(* Schneider Machine Expert - Basic project cel2_teste, file version 3.0.0.0 *)
(* ProjectInformations: Name=Novo projeto *)

HARDWARE
  Cpu 0: TM221CE16T
  ModuleExtensionObject 0: TM3DI16/G
  ModuleExtensionObject 1: TM3DQ16T/G
  ModuleExtensionObject 2: TM3DM8R/G
  ModuleExtensionObject 3: TM3DM8R/G
  ModuleExtensionObject 4: TM3DM8R/G
  ModuleExtensionObject 5: TM3SAF5R/G
  ModuleExtensionObject 6: TM3SAF5R/G
  EthernetConfiguration: NetworkName=M221, IpAllocationMode=FixedAddress, IpAddress=192.168.0.49, SubnetMask=255.255.255.0
  SerialLineConfiguration: Baud=Baud19200, Parity=ParityEven, DataBits=DataBits8, StopBits=StopBits1, PhysicalMedium=PhysicalMediumRs485, TransmissionMode=TransmissionModeModbusRtu, SlaveId=1, Addressing=SlaveAddressing
  MastTask: UsePeriodScanMode=false, PeriodScan=100
  FastTask: Period=255, FastTaskSubroutine=robo - clp
  CpuBehavior: StartingMode=StartAsPreviousState, AutoSaveRamOnEeprom=true, WatchdogPeriod=250

SYMBOLS  (address, symbol, comment, settings)
  %QWN300.9.0:X0 BIT1_SCADA
  %QWN300.9.0:X1 BIT2_SCADA
  %QWN300.9.0:X2 BIT3_SCADA
  %M0       M0  "primeiro paso - ligar celula"
  %M1       M1
  %M2       M2
  %M3       M3
  %M4       M4
  %M5       M5
  %M6       M6
  %M7       M7
  %M8       M8
  %M9       M9
  %M10      M10
  %M11      M11
  %M12      M12
  %M13      M13
  %M14      M14
  %M15      M15
  %M16      M16
  %M17      M17
  %M18      M18
  %M19      M19
  %M20      M20
  %M21      M21
  %M24      DESLIGA_BRANCO
  %M25      DESLIGA_CINZA
  %M26      DESLIGA_CINZA_ESCURO
  %M27      DESLIGA_PRETO
  %M28      DESLIGA_TRANSPARENTE
  %M32      ROBO_BRANCO
  %M33      ROBO_CINZA
  %M34      ROBO_CINZA_ESCURO
  %M35      ROBO_PRETO
  %M36      ROBO_TRANSPARENTE
  %M37      SCADA_SENSORESTEIRA
  %KW0      BASE_BRANCO  [Value=5]
  %KW1      BASE_CINZA  [Value=6]
  %KW2      BASE_CINZA_ESCURO  [Value=7]
  %KW3      BASE_PRETA  [Value=8]
  %KW4      BASE_TRANSPARENTE  [Value=9]
  %TM0      TIMER1  [Preset=4, Base=OneSecond]
  %TM1      TIMER2  [Preset=2, Base=OneSecond, IsRetentive=true]
  %TM2      TIMER3  [Preset=2, Base=OneSecond]
  %TM3      TIMER4  [Preset=2, Base=OneSecond]
  %TM4      TIMER5  [Preset=2, Base=OneSecond]
  %TM5      TIMER6  [Preset=2, Base=OneSecond]
  %TM6      TIMER7  [Preset=2, Base=OneSecond]
  %TM7      TIMER8  [Preset=5, Base=TenMilliSeconds]
  %TM8      TIMER9  [Preset=2, Base=OneSecond]
  %TM9      TIMER10  [Preset=2, Base=OneSecond]
  %TM10     TIMER11  [Preset=2, Base=OneSecond]
  %TM11     TIMER12  [Preset=2, Base=OneSecond]
  %TM12     TIMER13  [Preset=2, Base=OneSecond]
  %TM13     TIMERDESLIGA  [Preset=4, Base=OneSecond]
  %TM14     TIMERDESLIGA2  [Preset=4, Base=OneSecond]
  %TM15     TIMERDESLIGA3  [Preset=4, Base=OneSecond]
  %TM16     TIMERÚLTIMO  [Preset=4, Base=OneSecond]
  %TM17     TIMER17  [Preset=4, Base=OneSecond]
  %TM18     TIMER18  [Preset=2, Base=OneSecond]
  %TM19     TIMER19  [Preset=2, Base=OneSecond]
  %TM20     TIMER20  [Preset=2, Base=OneSecond]
  %TM21     TIMER21  [Preset=3, Base=OneSecond]
  %TM22     TIMER22  [Preset=2, Base=OneSecond]
  %TM23     TIMER23  [Preset=2, Base=OneSecond]
  %TM24       [Preset=1, Base=OneSecond]
  %TM25       [Preset=1, Base=OneSecond]
  %I0.0     RESET
  %I0.1     START_
  %I0.2     STOP
  %I0.3     PECA_ESTEIRA  "Sesnsor que detecta peçpa na garra na esteira"
  %I0.4     AVANCO_TRANSPARENTE  "Sensor Avanço Atuador Base Cinza Escuro"
  %I0.5     AVANCO_BRANCO  "Sensor Avanço Atuador Base Cinza"
  %I0.6     AVANCO_CINZA  "Sensor Avanço Atuador Base Transparente"
  %I0.7     AVANCO_CINZA_ESCURO  "Sensor Avanço Atuador Base Branco"
  %I0.8     AVANCO_PRETA  "Sensor Avanço Atuador Base Preta"
  %Q0.0     DISPENSER_PRETA  "Válvula Dispenser Preta"
  %Q0.1     DISPENSER_CINZA_ESCURO  "Válvula Dispenser Cinza escuro"
  %Q0.2     DISPENSER_CINZA  "Válvula Dispenser cinza claro"
  %Q0.3     DISPENSER_BRANCO  "Válvula Dispenser Branco"
  %Q0.4     DISPENSER_TRANSPARENTE  "Válvula Dispenser Transparente"
  %Q0.5     ATUADOR_X  "Válvula Atuador Eixo X"
  %Q0.6     ATUADOR_Z  "Válvula Atuador Eixo Z"
  %IN301.0.0   "Start forçado para a grob"  [Channel=START]
  %IN301.1.0   "Branco forçado GROB"  [Channel=BRANCO]
  %QN300.2.0 VENTOSA_SCADA  [Channel=NX3008_ventosa]
  %QN300.4.0   [Channel=NX3008_garra]
  %QN300.6.0 ATUADORX_SCADA  [Channel=NX3008_atuador_x]
  %QN300.7.0 ATUADORZ_SCADA  [Channel=NX3008_atuador_z]
  %IWN300.0.0 BASE_MODBUS  [Channel=NX3008_id_base]
  %IWN301.2.0 BASES_GROB  [Channel=Teste_bases]
  %QWN300.1.0   [Channel=NX3008_sensores]
  %QWN300.3.0   [Channel=NX3008_dispensers]
  %QWN300.5.0   [Channel=NX3008_sensor_garra_esteira]
  %QWN300.8.0 CORES  [Channel=NX3008_cores]
  %QWN300.9.0   [Channel=NX3008_Infos_robo]
  %I1.0     RECUOX  "sensor de recuo x"
  %I1.1     AVANCOX  "sensor de avanco x"
  %I1.2     RECUOZ  "sensor de recuo z"
  %I1.3     AVANCOZ  "sesnor de avanco z"
  %I1.4     GARRAABERTA  "sensor da garra aberta do atuador"
  %I1.5     SAIDADISPENSER  "sensor de presenca de saida do dispenser na garra do robo"
  %I1.6     GARRAABROB  "sensor de garra aberta do robo"
  %I1.14    OUTPUT1_VACUO
  %I1.15    OUTPUT2_RBG
  %Q2.0     ATUADORGARRA  "valvula da garra do atuador"
  %Q2.1     GARRAROB
  %Q2.3     VENTOSA_
  %I3.0     ENTRADA1  "modolo de io do robo sem enderecamento"
  %I3.1     ENTRADA2  "modolo de io do robo sem enderecamento"
  %I3.2     ROBOFINALIZADO
  %I3.3     LUZAMARELA
  %Q3.0     BIT1  "modolo de io do robo sem enderecamento"
  %Q3.1     BIT2  "modolo de io do robo sem enderecamento"
  %Q3.2     BIT3  "modolo de io do robo sem enderecamento"
  %I4.0       "Sensor de Recuo Eixo X - celula"
  %I4.1       "Sensor de Avanço Eixo X - esteira"
  %I4.2       "Sensor de Recuo Eixo Z - cima"
  %I4.3       "Sensor de Avanço Eixo Z - baixo"
  %Q4.0       "robo"
  %Q4.1       "robo"
  %Q4.2       "robo"
  %Q4.3       "robo"
  %I5.0       "Sensor de Garra Aberta"
  %I5.1       "Sensor de Peça Montagem"
  %I5.2       "Sensor de Presença Saida do Dispenser"
  %Q5.1       "Válvula Atuador Garra"
  %Q5.2       "vacuum generator"
  %Q5.3       "TORRE DE SINALIZAÇÃO"
  %I6.0     SA_OUTPUTON  "Saída de segurança ligada"
  %I6.1     SA_SUPPLY  "Fornecimento disponível (A1/A2)"
  %I6.2     SA_SUPPLYFAIL  "Fornecimento fora de tolerância"
  %I6.3     SA_CH1  "Canal 1 ativo"
  %I6.4     SA_CH2  "Canal 2 ativo"
  %I6.5     SA_START  "Início ativo"
  %I6.6     SA_K1  "Relé K1 ativado"
  %I6.7     SA_K2  "Relé k2 ativado"
  %I6.8       "Reserved"
  %I6.9     SA_S1  "S1 ativo"
  %I6.10    SA_S2  "S2 ativo"
  %I6.11    SA_S4  "S4 ativo"
  %I6.12    SA_WAITINGFORSTART  "Aguardando por condição de início"
  %I6.13      "Reserved"
  %Q6.0     SA_ENABLE  "Ativação das saídas de segurança habilitada"
  %Q6.1     SA_RESETMODULE  "Módulo de desativação (fonte atual desligada)"
  %Q6.2     SA_KEEPALIVE  "Função de segurança permanece ativa mesmo quando o barramento está 'inativo' (tempo esgotado)"
  %Q6.3       "Reserved"
  %I7.0     SA_OUTPUTON_0  "Saída de segurança ligada"
  %I7.1     SA_SUPPLY_0  "Fornecimento disponível (A1/A2)"
  %I7.2     SA_SUPPLYFAIL_0  "Fornecimento fora de tolerância"
  %I7.3     SA_CH1_0  "Canal 1 ativo"
  %I7.4     SA_CH2_0  "Canal 2 ativo"
  %I7.5     SA_START_0  "Início ativo"
  %I7.6     SA_K1_0  "Relé K1 ativado"
  %I7.7     SA_K2_0  "Relé k2 ativado"
  %I7.8       "Reserved"
  %I7.9     SA_S1_0  "S1 ativo"
  %I7.10    SA_S2_0  "S2 ativo"
  %I7.11    SA_S4_0  "S4 ativo"
  %I7.12    SA_WAITINGFORSTART_0  "Aguardando por condição de início"
  %I7.13      "Reserved"
  %Q7.0     SA_ENABLE_0  "Ativação das saídas de segurança habilitada"
  %Q7.1     SA_RESETMODULE_0  "Módulo de desativação (fonte atual desligada)"
  %Q7.2     SA_KEEPALIVE_0  "Função de segurança permanece ativa mesmo quando o barramento está 'inativo' (tempo esgotado)"
  %Q7.3       "Reserved"

POU Transferencia-SCADA
  (* SectionNumber=1 *)

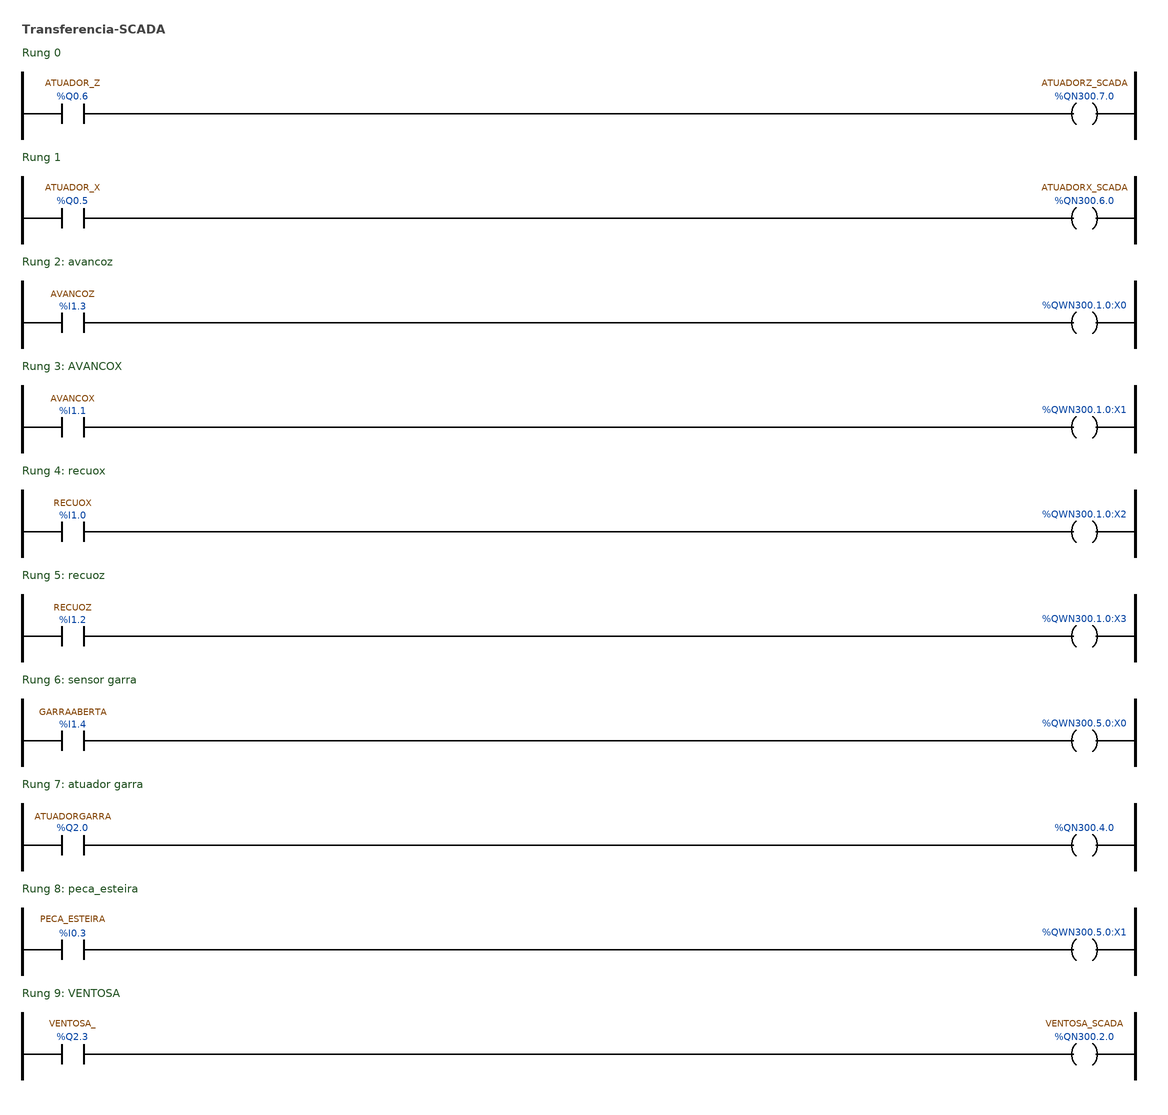

// Rung 0
  LD %Q0.6                (* ATUADOR_Z *)
  ST %QN300.7.0           (* ATUADORZ_SCADA *)
  // as ST:
  //   ATUADORZ_SCADA := ATUADOR_Z;

// Rung 1
  LD %Q0.5                (* ATUADOR_X *)
  ST %QN300.6.0           (* ATUADORX_SCADA *)
  // as ST:
  //   ATUADORX_SCADA := ATUADOR_X;

// Rung 2: avancoz
  LD %I1.3                (* AVANCOZ *)
  ST %QWN300.1.0:X0
  // as ST:
  //   %QWN300.1.0:X0 := AVANCOZ;

// Rung 3: AVANCOX
  LD %I1.1                (* AVANCOX *)
  ST %QWN300.1.0:X1
  // as ST:
  //   %QWN300.1.0:X1 := AVANCOX;

// Rung 4: recuox
  LD %I1.0                (* RECUOX *)
  ST %QWN300.1.0:X2
  // as ST:
  //   %QWN300.1.0:X2 := RECUOX;

// Rung 5: recuoz
  LD %I1.2                (* RECUOZ *)
  ST %QWN300.1.0:X3
  // as ST:
  //   %QWN300.1.0:X3 := RECUOZ;

// Rung 6: sensor garra
  LD %I1.4                (* GARRAABERTA *)
  ST %QWN300.5.0:X0
  // as ST:
  //   %QWN300.5.0:X0 := GARRAABERTA;

// Rung 7: atuador garra
  LD %Q2.0                (* ATUADORGARRA *)
  ST %QN300.4.0
  // as ST:
  //   %QN300.4.0 := ATUADORGARRA;

// Rung 8: peca_esteira
  LD %I0.3                (* PECA_ESTEIRA *)
  ST %QWN300.5.0:X1
  // as ST:
  //   %QWN300.5.0:X1 := PECA_ESTEIRA;

// Rung 9: VENTOSA
  LD %Q2.3                (* VENTOSA_ *)
  ST %QN300.2.0           (* VENTOSA_SCADA *)
  // as ST:
  //   VENTOSA_SCADA := VENTOSA_;

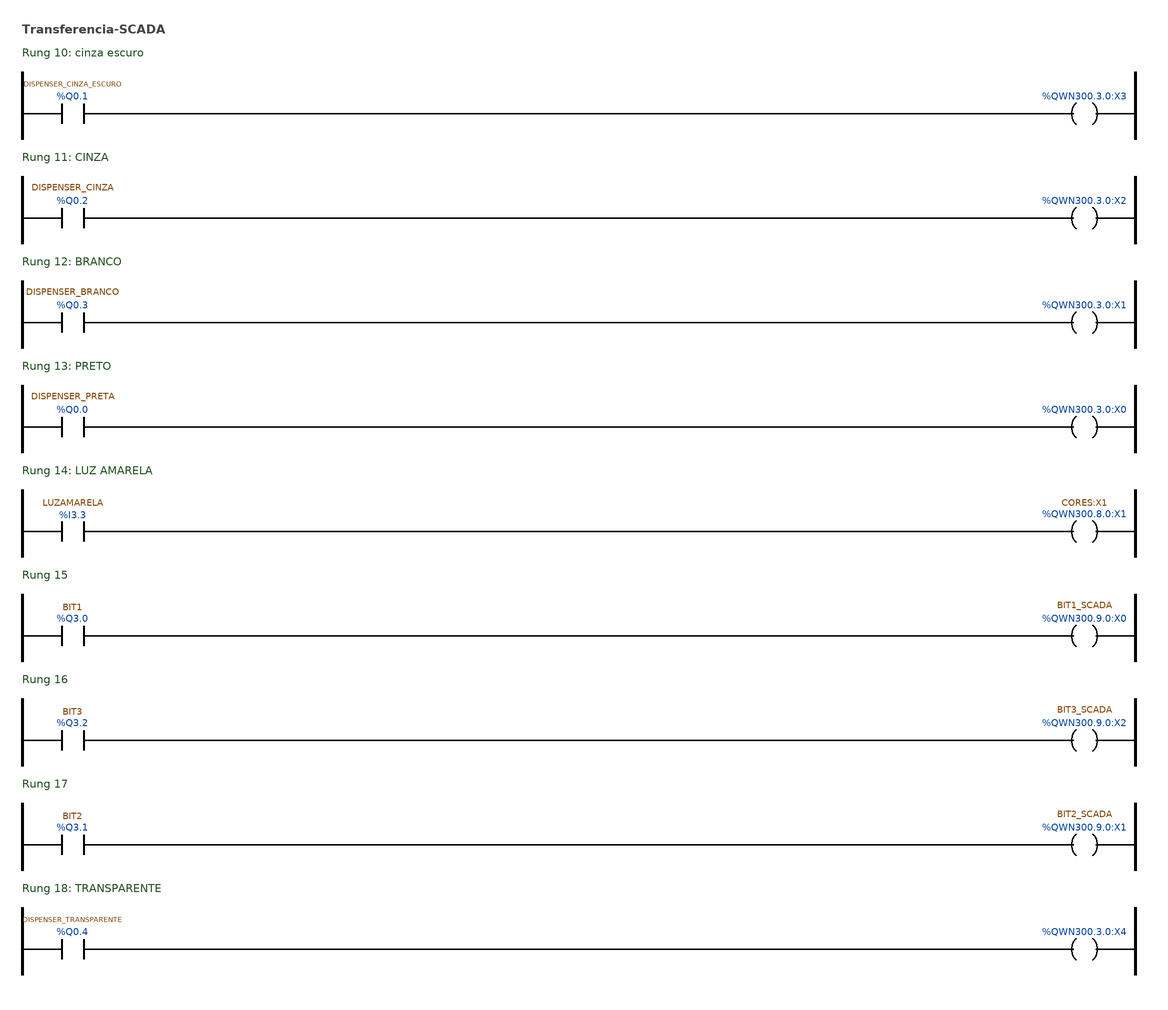

// Rung 10: cinza escuro
  LD %Q0.1                (* DISPENSER_CINZA_ESCURO *)
  ST %QWN300.3.0:X3
  // as ST:
  //   %QWN300.3.0:X3 := DISPENSER_CINZA_ESCURO;

// Rung 11: CINZA
  LD %Q0.2                (* DISPENSER_CINZA *)
  ST %QWN300.3.0:X2
  // as ST:
  //   %QWN300.3.0:X2 := DISPENSER_CINZA;

// Rung 12: BRANCO
  LD %Q0.3                (* DISPENSER_BRANCO *)
  ST %QWN300.3.0:X1
  // as ST:
  //   %QWN300.3.0:X1 := DISPENSER_BRANCO;

// Rung 13: PRETO
  LD %Q0.0                (* DISPENSER_PRETA *)
  ST %QWN300.3.0:X0
  // as ST:
  //   %QWN300.3.0:X0 := DISPENSER_PRETA;

// Rung 14: LUZ AMARELA
  LD %I3.3                (* LUZAMARELA *)
  ST %QWN300.8.0:X1       (* CORES *)
  // as ST:
  //   CORES:X1 := LUZAMARELA;

// Rung 15
  LD %Q3.0                (* BIT1 *)
  ST %QWN300.9.0:X0
  // as ST:
  //   %QWN300.9.0:X0 := BIT1;

// Rung 16
  LD %Q3.2                (* BIT3 *)
  ST %QWN300.9.0:X2
  // as ST:
  //   %QWN300.9.0:X2 := BIT3;

// Rung 17
  LD %Q3.1                (* BIT2 *)
  ST %QWN300.9.0:X1
  // as ST:
  //   %QWN300.9.0:X1 := BIT2;

// Rung 18: TRANSPARENTE
  LD %Q0.4                (* DISPENSER_TRANSPARENTE *)
  ST %QWN300.3.0:X4
  // as ST:
  //   %QWN300.3.0:X4 := DISPENSER_TRANSPARENTE;

POU celula 2
  (* SectionNumber=2 *)

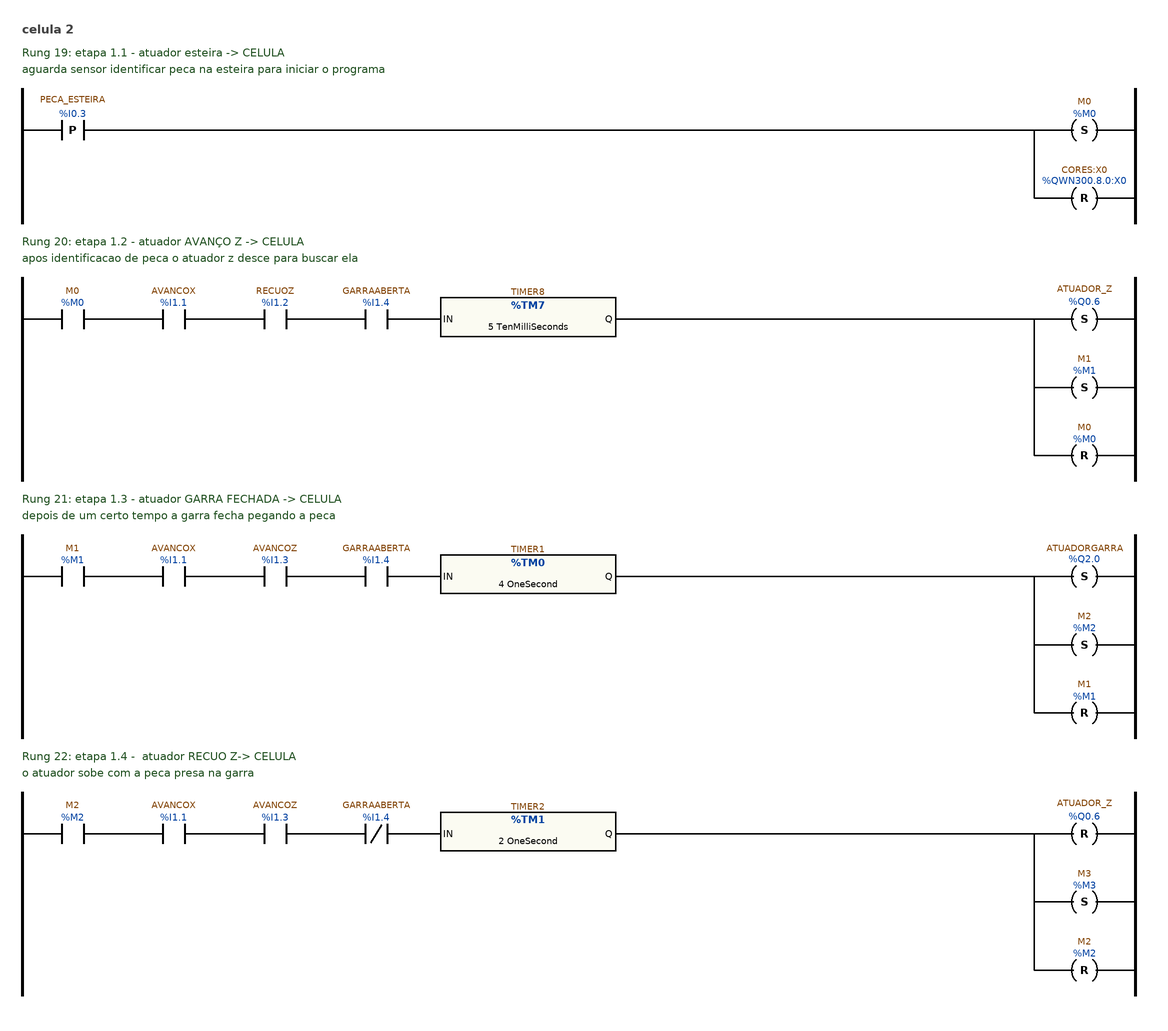

// Rung 19: etapa 1.1 - atuador esteira -> CELULA
// aguarda sensor identificar peca na esteira para iniciar o programa
  LDR %I0.3               (* PECA_ESTEIRA *)
  S %M0                   (* M0 *)
  R %QWN300.8.0:X0        (* CORES *)
  // as ST:
  //   IF RISING(PECA_ESTEIRA) THEN M0 := TRUE; END_IF;
  //   IF RISING(PECA_ESTEIRA) THEN CORES:X0 := FALSE; END_IF;

// Rung 20: etapa 1.2 - atuador AVANÇO Z -> CELULA
// apos identificacao de peca o atuador z desce para buscar ela
  BLK %TM7                (* TIMER8 *)
  LD %M0                  (* M0 *)
  AND %I1.1               (* AVANCOX *)
  AND %I1.2               (* RECUOZ *)
  AND %I1.4               (* GARRAABERTA *)
  IN
  OUT_BLK
  LD Q
  S %Q0.6                 (* ATUADOR_Z *)
  S %M1                   (* M1 *)
  R %M0                   (* M0 *)
  END_BLK
  // as ST:
  //   TIMER8(IN := M0 AND AVANCOX AND RECUOZ AND GARRAABERTA);
  //   IF TIMER8.Q THEN ATUADOR_Z := TRUE; END_IF;
  //   IF TIMER8.Q THEN M1 := TRUE; END_IF;
  //   IF TIMER8.Q THEN M0 := FALSE; END_IF;

// Rung 21: etapa 1.3 - atuador GARRA FECHADA -> CELULA
// depois de um certo tempo a garra fecha pegando a peca
  BLK %TM0                (* TIMER1 *)
  LD %M1                  (* M1 *)
  AND %I1.1               (* AVANCOX *)
  AND %I1.3               (* AVANCOZ *)
  AND %I1.4               (* GARRAABERTA *)
  IN
  OUT_BLK
  LD Q
  S %Q2.0                 (* ATUADORGARRA *)
  S %M2                   (* M2 *)
  R %M1                   (* M1 *)
  END_BLK
  // as ST:
  //   TIMER1(IN := M1 AND AVANCOX AND AVANCOZ AND GARRAABERTA);
  //   IF TIMER1.Q THEN ATUADORGARRA := TRUE; END_IF;
  //   IF TIMER1.Q THEN M2 := TRUE; END_IF;
  //   IF TIMER1.Q THEN M1 := FALSE; END_IF;

// Rung 22: etapa 1.4 -  atuador RECUO Z-> CELULA
// o atuador sobe com a peca presa na garra
  BLK %TM1                (* TIMER2 *)
  LD %M2                  (* M2 *)
  AND %I1.1               (* AVANCOX *)
  AND %I1.3               (* AVANCOZ *)
  ANDN %I1.4              (* GARRAABERTA *)
  IN
  OUT_BLK
  LD Q
  R %Q0.6                 (* ATUADOR_Z *)
  S %M3                   (* M3 *)
  R %M2                   (* M2 *)
  END_BLK
  // as ST:
  //   TIMER2(IN := M2 AND AVANCOX AND AVANCOZ AND NOT GARRAABERTA);
  //   IF TIMER2.Q THEN ATUADOR_Z := FALSE; END_IF;
  //   IF TIMER2.Q THEN M3 := TRUE; END_IF;
  //   IF TIMER2.Q THEN M2 := FALSE; END_IF;

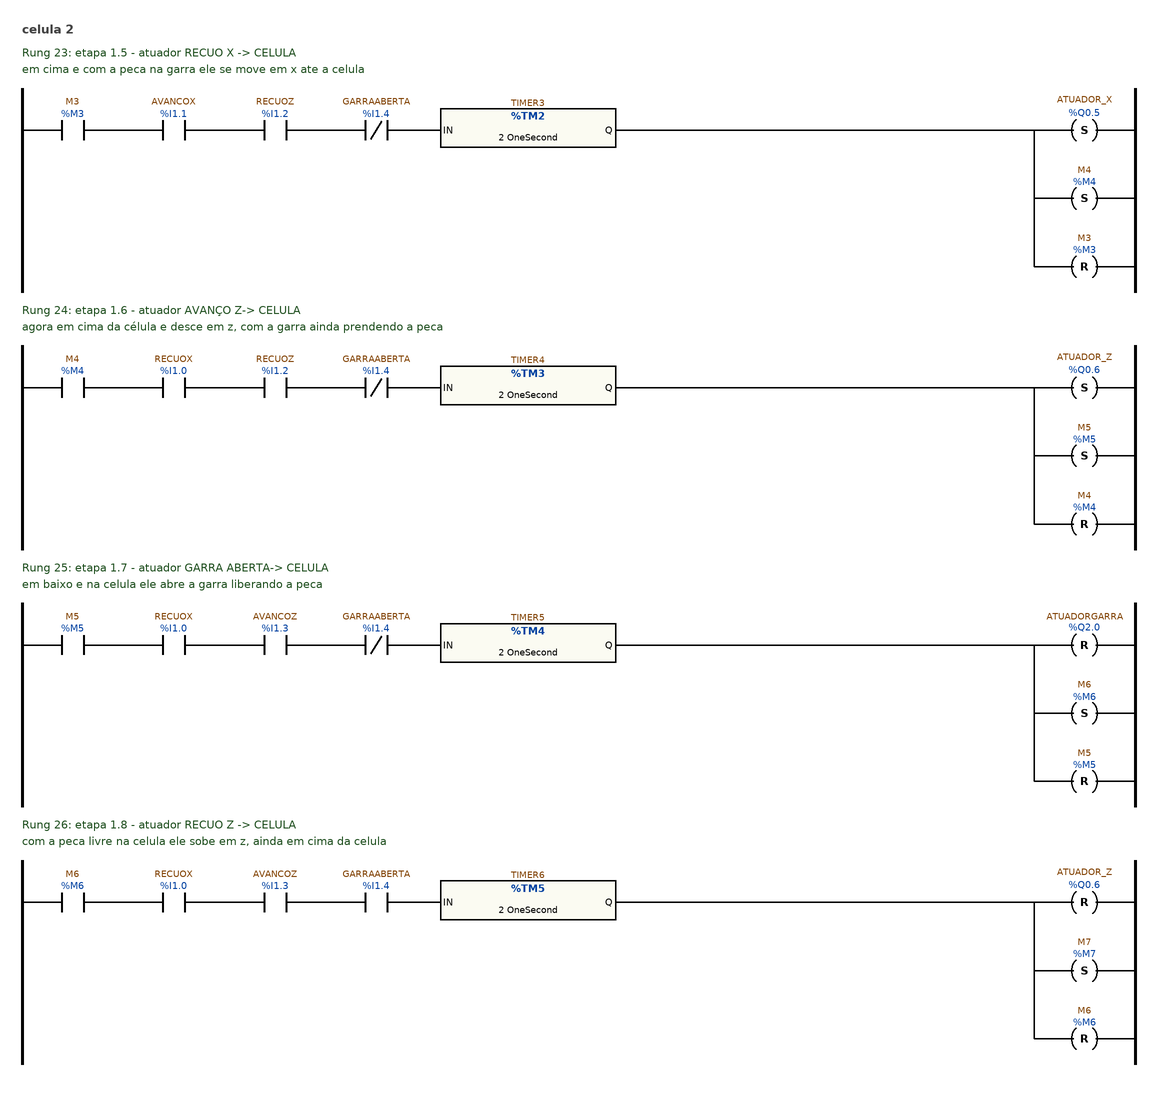

// Rung 23: etapa 1.5 - atuador RECUO X -> CELULA
// em cima e com a peca na garra ele se move em x ate a celula
  BLK %TM2                (* TIMER3 *)
  LD %M3                  (* M3 *)
  AND %I1.1               (* AVANCOX *)
  AND %I1.2               (* RECUOZ *)
  ANDN %I1.4              (* GARRAABERTA *)
  IN
  OUT_BLK
  LD Q
  S %Q0.5                 (* ATUADOR_X *)
  S %M4                   (* M4 *)
  R %M3                   (* M3 *)
  END_BLK
  // as ST:
  //   TIMER3(IN := M3 AND AVANCOX AND RECUOZ AND NOT GARRAABERTA);
  //   IF TIMER3.Q THEN ATUADOR_X := TRUE; END_IF;
  //   IF TIMER3.Q THEN M4 := TRUE; END_IF;
  //   IF TIMER3.Q THEN M3 := FALSE; END_IF;

// Rung 24: etapa 1.6 - atuador AVANÇO Z-> CELULA
// agora em cima da célula e desce em z, com a garra ainda prendendo a peca
  BLK %TM3                (* TIMER4 *)
  LD %M4                  (* M4 *)
  AND %I1.0               (* RECUOX *)
  AND %I1.2               (* RECUOZ *)
  ANDN %I1.4              (* GARRAABERTA *)
  IN
  OUT_BLK
  LD Q
  S %Q0.6                 (* ATUADOR_Z *)
  S %M5                   (* M5 *)
  R %M4                   (* M4 *)
  END_BLK
  // as ST:
  //   TIMER4(IN := M4 AND RECUOX AND RECUOZ AND NOT GARRAABERTA);
  //   IF TIMER4.Q THEN ATUADOR_Z := TRUE; END_IF;
  //   IF TIMER4.Q THEN M5 := TRUE; END_IF;
  //   IF TIMER4.Q THEN M4 := FALSE; END_IF;

// Rung 25: etapa 1.7 - atuador GARRA ABERTA-> CELULA
// em baixo e na celula ele abre a garra liberando a peca
  BLK %TM4                (* TIMER5 *)
  LD %M5                  (* M5 *)
  AND %I1.0               (* RECUOX *)
  AND %I1.3               (* AVANCOZ *)
  ANDN %I1.4              (* GARRAABERTA *)
  IN
  OUT_BLK
  LD Q
  R %Q2.0                 (* ATUADORGARRA *)
  S %M6                   (* M6 *)
  R %M5                   (* M5 *)
  END_BLK
  // as ST:
  //   TIMER5(IN := M5 AND RECUOX AND AVANCOZ AND NOT GARRAABERTA);
  //   IF TIMER5.Q THEN ATUADORGARRA := FALSE; END_IF;
  //   IF TIMER5.Q THEN M6 := TRUE; END_IF;
  //   IF TIMER5.Q THEN M5 := FALSE; END_IF;

// Rung 26: etapa 1.8 - atuador RECUO Z -> CELULA
// com a peca livre na celula ele sobe em z, ainda em cima da celula
  BLK %TM5                (* TIMER6 *)
  LD %M6                  (* M6 *)
  AND %I1.0               (* RECUOX *)
  AND %I1.3               (* AVANCOZ *)
  AND %I1.4               (* GARRAABERTA *)
  IN
  OUT_BLK
  LD Q
  R %Q0.6                 (* ATUADOR_Z *)
  S %M7                   (* M7 *)
  R %M6                   (* M6 *)
  END_BLK
  // as ST:
  //   TIMER6(IN := M6 AND RECUOX AND AVANCOZ AND GARRAABERTA);
  //   IF TIMER6.Q THEN ATUADOR_Z := FALSE; END_IF;
  //   IF TIMER6.Q THEN M7 := TRUE; END_IF;
  //   IF TIMER6.Q THEN M6 := FALSE; END_IF;

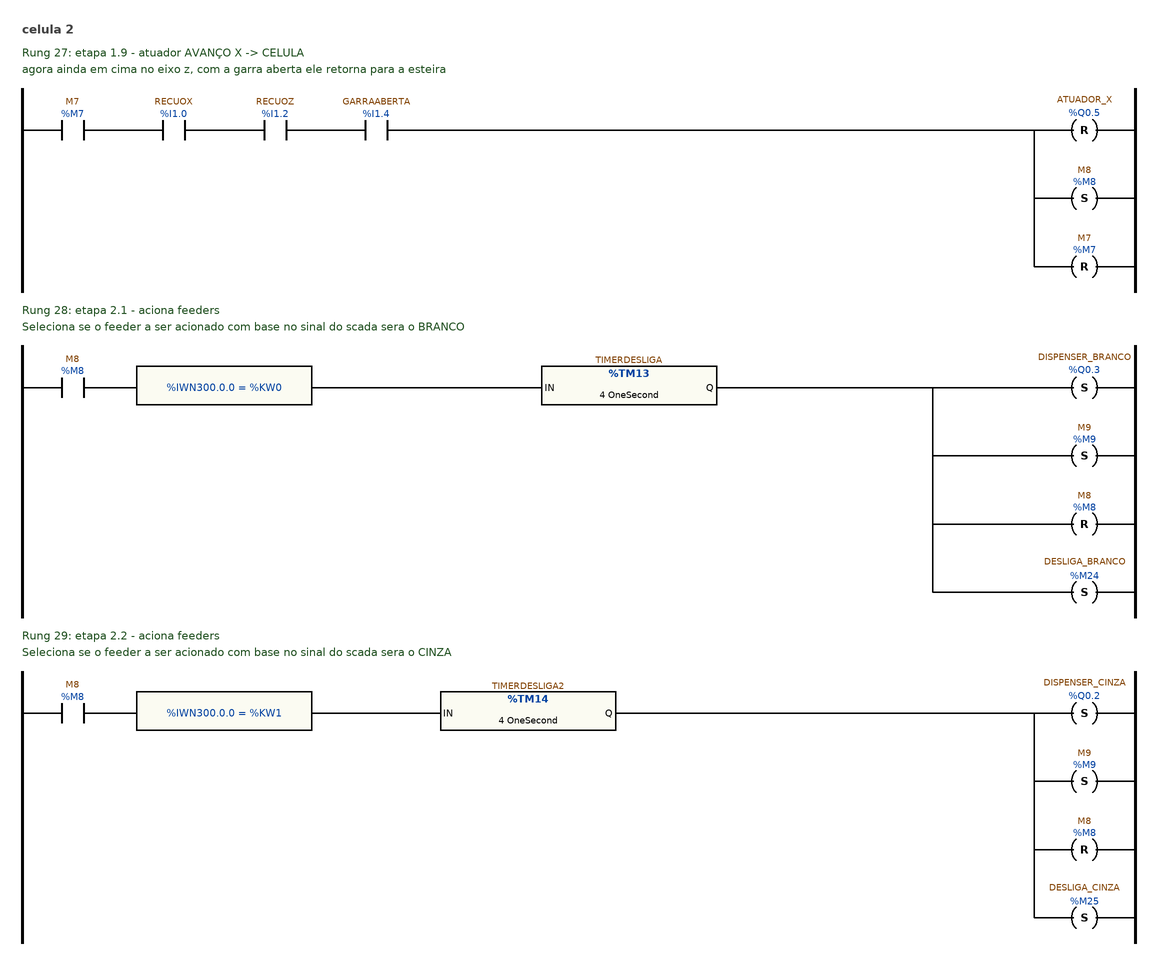

// Rung 27: etapa 1.9 - atuador AVANÇO X -> CELULA
// agora ainda em cima no eixo z, com a garra aberta ele retorna para a esteira
  LD %M7                  (* M7 *)
  AND %I1.0               (* RECUOX *)
  AND %I1.2               (* RECUOZ *)
  AND %I1.4               (* GARRAABERTA *)
  R %Q0.5                 (* ATUADOR_X *)
  S %M8                   (* M8 *)
  R %M7                   (* M7 *)
  // as ST:
  //   IF M7 AND RECUOX AND RECUOZ AND GARRAABERTA THEN ATUADOR_X := FALSE; END_IF;
  //   IF M7 AND RECUOX AND RECUOZ AND GARRAABERTA THEN M8 := TRUE; END_IF;
  //   IF M7 AND RECUOX AND RECUOZ AND GARRAABERTA THEN M7 := FALSE; END_IF;

// Rung 28: etapa 2.1 - aciona feeders
// Seleciona se o feeder a ser acionado com base no sinal do scada sera o BRANCO
  BLK %TM13               (* TIMERDESLIGA *)
  LD %M8                  (* M8 *)
  AND [ %IWN300.0.0 = %KW0 ](* BASE_MODBUS, BASE_BRANCO *)
  IN
  OUT_BLK
  LD Q
  S %Q0.3                 (* DISPENSER_BRANCO *)
  S %M9                   (* M9 *)
  R %M8                   (* M8 *)
  S %M24                  (* DESLIGA_BRANCO *)
  END_BLK
  // as ST:
  //   TIMERDESLIGA(IN := M8 AND BASE_MODBUS = BASE_BRANCO);
  //   IF TIMERDESLIGA.Q THEN DISPENSER_BRANCO := TRUE; END_IF;
  //   IF TIMERDESLIGA.Q THEN M9 := TRUE; END_IF;
  //   IF TIMERDESLIGA.Q THEN M8 := FALSE; END_IF;
  //   IF TIMERDESLIGA.Q THEN DESLIGA_BRANCO := TRUE; END_IF;

// Rung 29: etapa 2.2 - aciona feeders
// Seleciona se o feeder a ser acionado com base no sinal do scada sera o CINZA
  BLK %TM14               (* TIMERDESLIGA2 *)
  LD %M8                  (* M8 *)
  AND [ %IWN300.0.0 = %KW1 ](* BASE_MODBUS, BASE_CINZA *)
  IN
  OUT_BLK
  LD Q
  S %Q0.2                 (* DISPENSER_CINZA *)
  S %M9                   (* M9 *)
  R %M8                   (* M8 *)
  S %M25                  (* DESLIGA_CINZA *)
  END_BLK
  // as ST:
  //   TIMERDESLIGA2(IN := M8 AND BASE_MODBUS = BASE_CINZA);
  //   IF TIMERDESLIGA2.Q THEN DISPENSER_CINZA := TRUE; END_IF;
  //   IF TIMERDESLIGA2.Q THEN M9 := TRUE; END_IF;
  //   IF TIMERDESLIGA2.Q THEN M8 := FALSE; END_IF;
  //   IF TIMERDESLIGA2.Q THEN DESLIGA_CINZA := TRUE; END_IF;

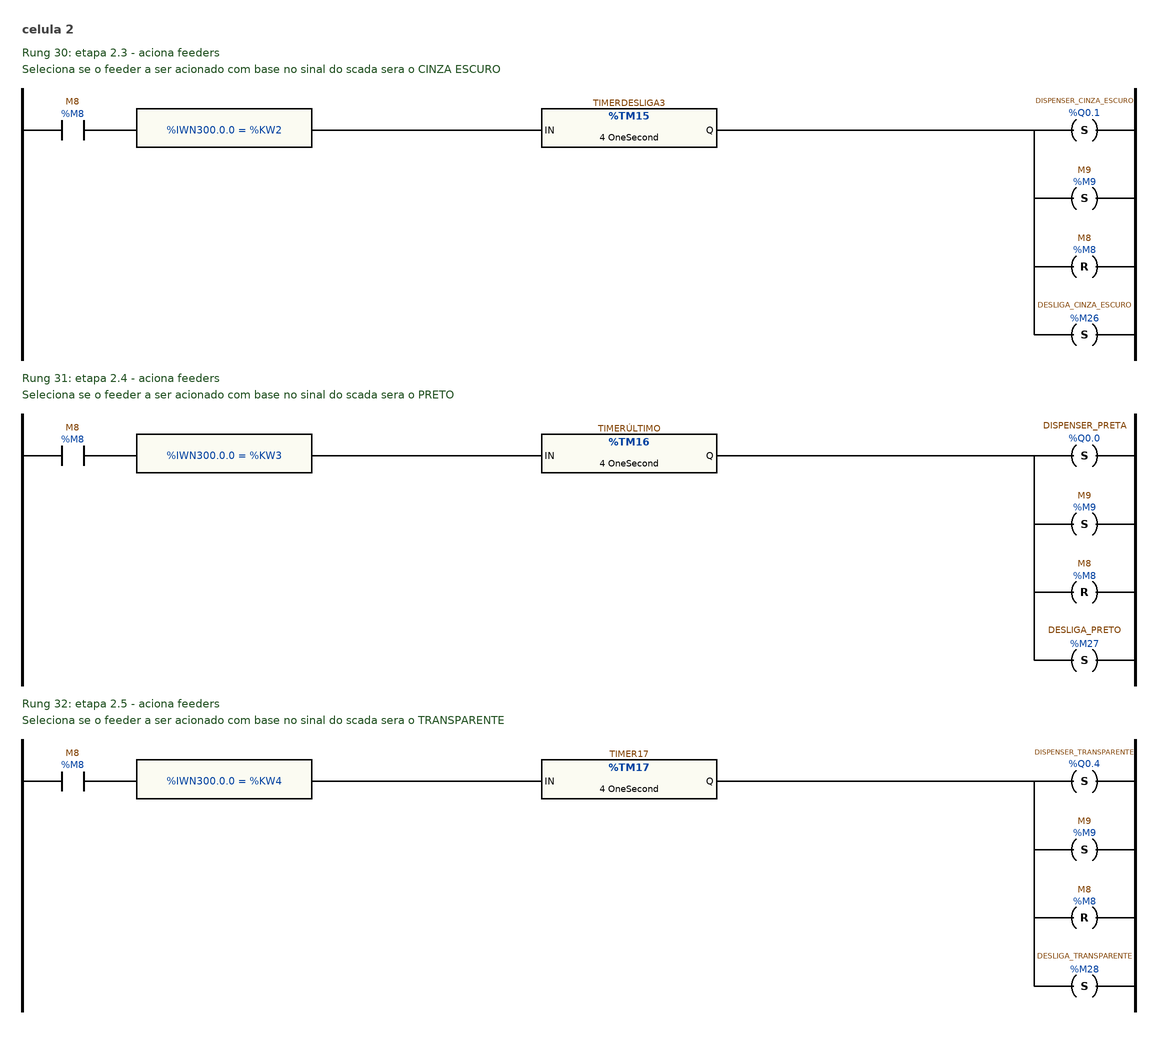

// Rung 30: etapa 2.3 - aciona feeders
// Seleciona se o feeder a ser acionado com base no sinal do scada sera o CINZA ESCURO
  BLK %TM15               (* TIMERDESLIGA3 *)
  LD %M8                  (* M8 *)
  AND [ %IWN300.0.0 = %KW2 ](* BASE_MODBUS, BASE_CINZA_ESCURO *)
  IN
  OUT_BLK
  LD Q
  S %Q0.1                 (* DISPENSER_CINZA_ESCURO *)
  S %M9                   (* M9 *)
  R %M8                   (* M8 *)
  S %M26                  (* DESLIGA_CINZA_ESCURO *)
  END_BLK
  // as ST:
  //   TIMERDESLIGA3(IN := M8 AND BASE_MODBUS = BASE_CINZA_ESCURO);
  //   IF TIMERDESLIGA3.Q THEN DISPENSER_CINZA_ESCURO := TRUE; END_IF;
  //   IF TIMERDESLIGA3.Q THEN M9 := TRUE; END_IF;
  //   IF TIMERDESLIGA3.Q THEN M8 := FALSE; END_IF;
  //   IF TIMERDESLIGA3.Q THEN DESLIGA_CINZA_ESCURO := TRUE; END_IF;

// Rung 31: etapa 2.4 - aciona feeders
// Seleciona se o feeder a ser acionado com base no sinal do scada sera o PRETO
  BLK %TM16               (* TIMERÚLTIMO *)
  LD %M8                  (* M8 *)
  AND [ %IWN300.0.0 = %KW3 ](* BASE_MODBUS, BASE_PRETA *)
  IN
  OUT_BLK
  LD Q
  S %Q0.0                 (* DISPENSER_PRETA *)
  S %M9                   (* M9 *)
  R %M8                   (* M8 *)
  S %M27                  (* DESLIGA_PRETO *)
  END_BLK
  // as ST:
  //   TIMERÚLTIMO(IN := M8 AND BASE_MODBUS = BASE_PRETA);
  //   IF TIMERÚLTIMO.Q THEN DISPENSER_PRETA := TRUE; END_IF;
  //   IF TIMERÚLTIMO.Q THEN M9 := TRUE; END_IF;
  //   IF TIMERÚLTIMO.Q THEN M8 := FALSE; END_IF;
  //   IF TIMERÚLTIMO.Q THEN DESLIGA_PRETO := TRUE; END_IF;

// Rung 32: etapa 2.5 - aciona feeders
// Seleciona se o feeder a ser acionado com base no sinal do scada sera o TRANSPARENTE
  BLK %TM17               (* TIMER17 *)
  LD %M8                  (* M8 *)
  AND [ %IWN300.0.0 = %KW4 ](* BASE_MODBUS, BASE_TRANSPARENTE *)
  IN
  OUT_BLK
  LD Q
  S %Q0.4                 (* DISPENSER_TRANSPARENTE *)
  S %M9                   (* M9 *)
  R %M8                   (* M8 *)
  S %M28                  (* DESLIGA_TRANSPARENTE *)
  END_BLK
  // as ST:
  //   TIMER17(IN := M8 AND BASE_MODBUS = BASE_TRANSPARENTE);
  //   IF TIMER17.Q THEN DISPENSER_TRANSPARENTE := TRUE; END_IF;
  //   IF TIMER17.Q THEN M9 := TRUE; END_IF;
  //   IF TIMER17.Q THEN M8 := FALSE; END_IF;
  //   IF TIMER17.Q THEN DESLIGA_TRANSPARENTE := TRUE; END_IF;

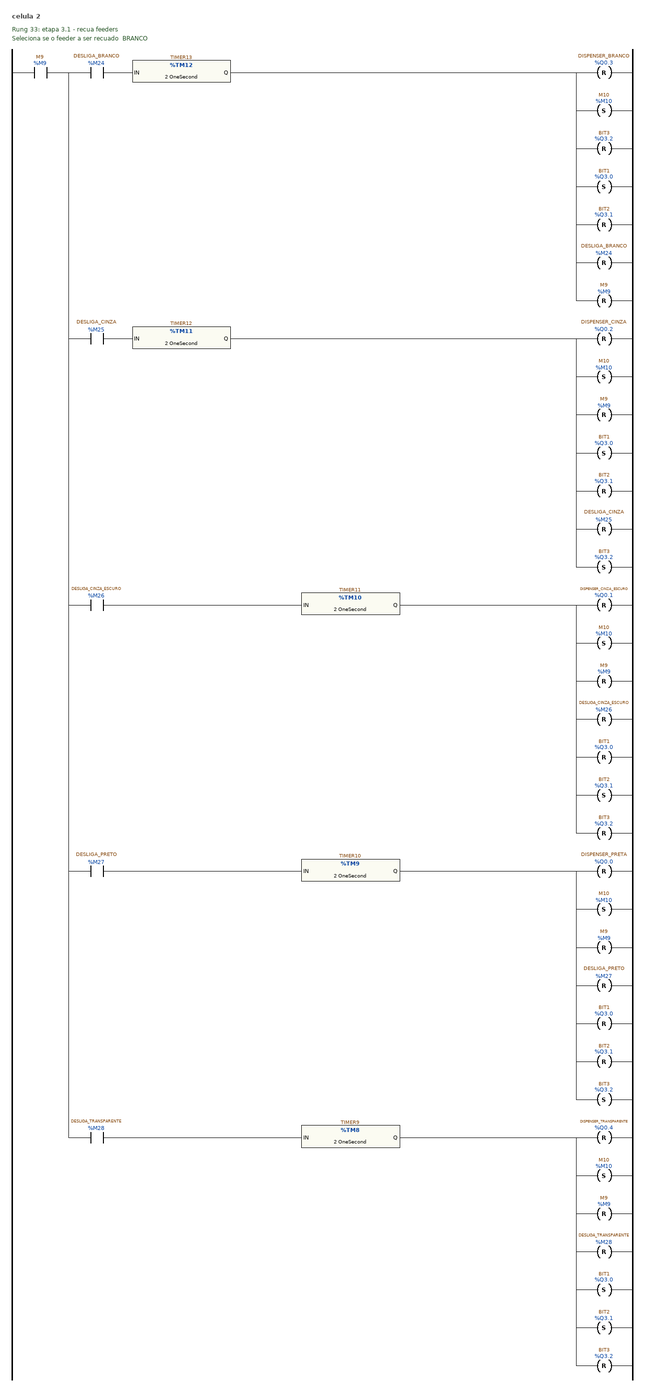

// Rung 33: etapa 3.1 - recua feeders
// Seleciona se o feeder a ser recuado  BRANCO
  LD 1
  MULTIFB
  LD 1
  AND %M9                 (* M9 *)
  ST %MW2009:X0
  BLK %TM12               (* TIMER13 *)
  LD %MW2009:X0
  AND %M24                (* DESLIGA_BRANCO *)
  IN
  OUT_BLK
  LD Q
  R %Q0.3                 (* DISPENSER_BRANCO *)
  S %M10                  (* M10 *)
  R %Q3.2                 (* BIT3 *)
  S %Q3.0                 (* BIT1 *)
  R %Q3.1                 (* BIT2 *)
  R %M24                  (* DESLIGA_BRANCO *)
  R %M9                   (* M9 *)
  END_BLK
  BLK %TM11               (* TIMER12 *)
  LD %MW2009:X0
  AND %M25                (* DESLIGA_CINZA *)
  IN
  OUT_BLK
  LD Q
  R %Q0.2                 (* DISPENSER_CINZA *)
  S %M10                  (* M10 *)
  R %M9                   (* M9 *)
  S %Q3.0                 (* BIT1 *)
  R %Q3.1                 (* BIT2 *)
  R %M25                  (* DESLIGA_CINZA *)
  S %Q3.2                 (* BIT3 *)
  END_BLK
  BLK %TM10               (* TIMER11 *)
  LD %MW2009:X0
  AND %M26                (* DESLIGA_CINZA_ESCURO *)
  IN
  OUT_BLK
  LD Q
  R %Q0.1                 (* DISPENSER_CINZA_ESCURO *)
  S %M10                  (* M10 *)
  R %M9                   (* M9 *)
  R %M26                  (* DESLIGA_CINZA_ESCURO *)
  R %Q3.0                 (* BIT1 *)
  S %Q3.1                 (* BIT2 *)
  R %Q3.2                 (* BIT3 *)
  END_BLK
  BLK %TM9                (* TIMER10 *)
  LD %MW2009:X0
  AND %M27                (* DESLIGA_PRETO *)
  IN
  OUT_BLK
  LD Q
  R %Q0.0                 (* DISPENSER_PRETA *)
  S %M10                  (* M10 *)
  R %M9                   (* M9 *)
  R %M27                  (* DESLIGA_PRETO *)
  R %Q3.0                 (* BIT1 *)
  R %Q3.1                 (* BIT2 *)
  S %Q3.2                 (* BIT3 *)
  END_BLK
  BLK %TM8                (* TIMER9 *)
  LD %MW2009:X0
  AND %M28                (* DESLIGA_TRANSPARENTE *)
  IN
  OUT_BLK
  LD Q
  R %Q0.4                 (* DISPENSER_TRANSPARENTE *)
  S %M10                  (* M10 *)
  R %M9                   (* M9 *)
  R %M28                  (* DESLIGA_TRANSPARENTE *)
  S %Q3.0                 (* BIT1 *)
  S %Q3.1                 (* BIT2 *)
  R %Q3.2                 (* BIT3 *)
  END_BLK
  MULTIFB
  // as ST:
  //   TIMER13(IN := M9 AND DESLIGA_BRANCO);
  //   IF TIMER13.Q THEN DISPENSER_BRANCO := FALSE; END_IF;
  //   IF TIMER13.Q THEN M10 := TRUE; END_IF;
  //   IF TIMER13.Q THEN BIT3 := FALSE; END_IF;
  //   IF TIMER13.Q THEN BIT1 := TRUE; END_IF;
  //   IF TIMER13.Q THEN BIT2 := FALSE; END_IF;
  //   IF TIMER13.Q THEN DESLIGA_BRANCO := FALSE; END_IF;
  //   _t1 := M9;
  //   IF TIMER13.Q THEN M9 := FALSE; END_IF;
  //   TIMER12(IN := _t1 AND DESLIGA_CINZA);
  //   IF TIMER12.Q THEN DISPENSER_CINZA := FALSE; END_IF;
  //   IF TIMER12.Q THEN M10 := TRUE; END_IF;
  //   IF TIMER12.Q THEN M9 := FALSE; END_IF;
  //   IF TIMER12.Q THEN BIT1 := TRUE; END_IF;
  //   IF TIMER12.Q THEN BIT2 := FALSE; END_IF;
  //   IF TIMER12.Q THEN DESLIGA_CINZA := FALSE; END_IF;
  //   IF TIMER12.Q THEN BIT3 := TRUE; END_IF;
  //   TIMER11(IN := _t1 AND DESLIGA_CINZA_ESCURO);
  //   IF TIMER11.Q THEN DISPENSER_CINZA_ESCURO := FALSE; END_IF;
  //   IF TIMER11.Q THEN M10 := TRUE; END_IF;
  //   IF TIMER11.Q THEN M9 := FALSE; END_IF;
  //   IF TIMER11.Q THEN DESLIGA_CINZA_ESCURO := FALSE; END_IF;
  //   IF TIMER11.Q THEN BIT1 := FALSE; END_IF;
  //   IF TIMER11.Q THEN BIT2 := TRUE; END_IF;
  //   IF TIMER11.Q THEN BIT3 := FALSE; END_IF;
  //   TIMER10(IN := _t1 AND DESLIGA_PRETO);
  //   IF TIMER10.Q THEN DISPENSER_PRETA := FALSE; END_IF;
  //   IF TIMER10.Q THEN M10 := TRUE; END_IF;
  //   IF TIMER10.Q THEN M9 := FALSE; END_IF;
  //   IF TIMER10.Q THEN DESLIGA_PRETO := FALSE; END_IF;
  //   IF TIMER10.Q THEN BIT1 := FALSE; END_IF;
  //   IF TIMER10.Q THEN BIT2 := FALSE; END_IF;
  //   IF TIMER10.Q THEN BIT3 := TRUE; END_IF;
  //   TIMER9(IN := _t1 AND DESLIGA_TRANSPARENTE);
  //   IF TIMER9.Q THEN DISPENSER_TRANSPARENTE := FALSE; END_IF;
  //   IF TIMER9.Q THEN M10 := TRUE; END_IF;
  //   IF TIMER9.Q THEN M9 := FALSE; END_IF;
  //   IF TIMER9.Q THEN DESLIGA_TRANSPARENTE := FALSE; END_IF;
  //   IF TIMER9.Q THEN BIT1 := TRUE; END_IF;
  //   IF TIMER9.Q THEN BIT2 := TRUE; END_IF;
  //   IF TIMER9.Q THEN BIT3 := FALSE; END_IF;

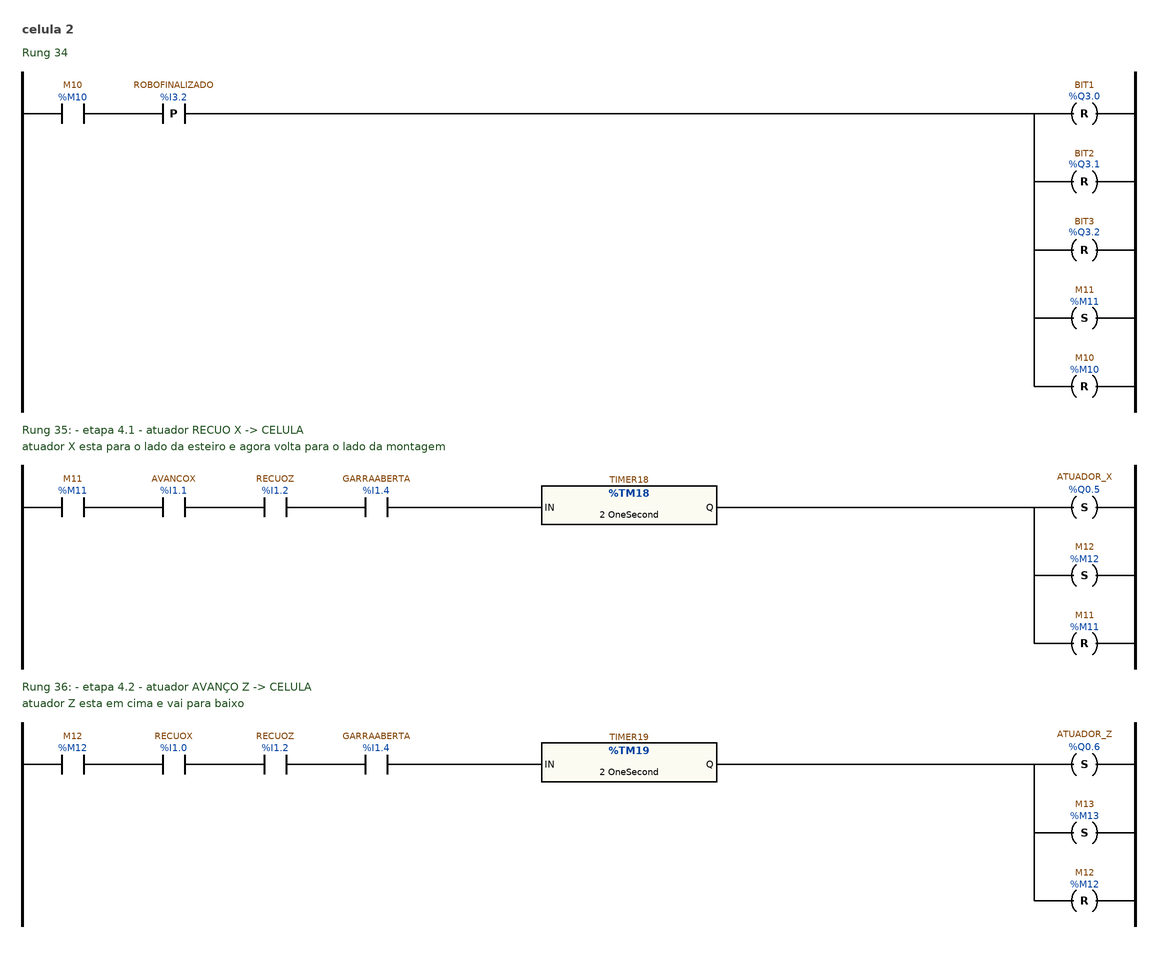

// Rung 34
  LD %M10                 (* M10 *)
  ANDR %I3.2              (* ROBOFINALIZADO *)
  R %Q3.0                 (* BIT1 *)
  R %Q3.1                 (* BIT2 *)
  R %Q3.2                 (* BIT3 *)
  S %M11                  (* M11 *)
  R %M10                  (* M10 *)
  // as ST:
  //   IF M10 AND RISING(ROBOFINALIZADO) THEN BIT1 := FALSE; END_IF;
  //   IF M10 AND RISING(ROBOFINALIZADO) THEN BIT2 := FALSE; END_IF;
  //   IF M10 AND RISING(ROBOFINALIZADO) THEN BIT3 := FALSE; END_IF;
  //   IF M10 AND RISING(ROBOFINALIZADO) THEN M11 := TRUE; END_IF;
  //   IF M10 AND RISING(ROBOFINALIZADO) THEN M10 := FALSE; END_IF;

// Rung 35: - etapa 4.1 - atuador RECUO X -> CELULA
// atuador X esta para o lado da esteiro e agora volta para o lado da montagem
  BLK %TM18               (* TIMER18 *)
  LD %M11                 (* M11 *)
  AND %I1.1               (* AVANCOX *)
  AND %I1.2               (* RECUOZ *)
  AND %I1.4               (* GARRAABERTA *)
  IN
  OUT_BLK
  LD Q
  S %Q0.5                 (* ATUADOR_X *)
  S %M12                  (* M12 *)
  R %M11                  (* M11 *)
  END_BLK
  // as ST:
  //   TIMER18(IN := M11 AND AVANCOX AND RECUOZ AND GARRAABERTA);
  //   IF TIMER18.Q THEN ATUADOR_X := TRUE; END_IF;
  //   IF TIMER18.Q THEN M12 := TRUE; END_IF;
  //   IF TIMER18.Q THEN M11 := FALSE; END_IF;

// Rung 36: - etapa 4.2 - atuador AVANÇO Z -> CELULA
// atuador Z esta em cima e vai para baixo
  BLK %TM19               (* TIMER19 *)
  LD %M12                 (* M12 *)
  AND %I1.0               (* RECUOX *)
  AND %I1.2               (* RECUOZ *)
  AND %I1.4               (* GARRAABERTA *)
  IN
  OUT_BLK
  LD Q
  S %Q0.6                 (* ATUADOR_Z *)
  S %M13                  (* M13 *)
  R %M12                  (* M12 *)
  END_BLK
  // as ST:
  //   TIMER19(IN := M12 AND RECUOX AND RECUOZ AND GARRAABERTA);
  //   IF TIMER19.Q THEN ATUADOR_Z := TRUE; END_IF;
  //   IF TIMER19.Q THEN M13 := TRUE; END_IF;
  //   IF TIMER19.Q THEN M12 := FALSE; END_IF;

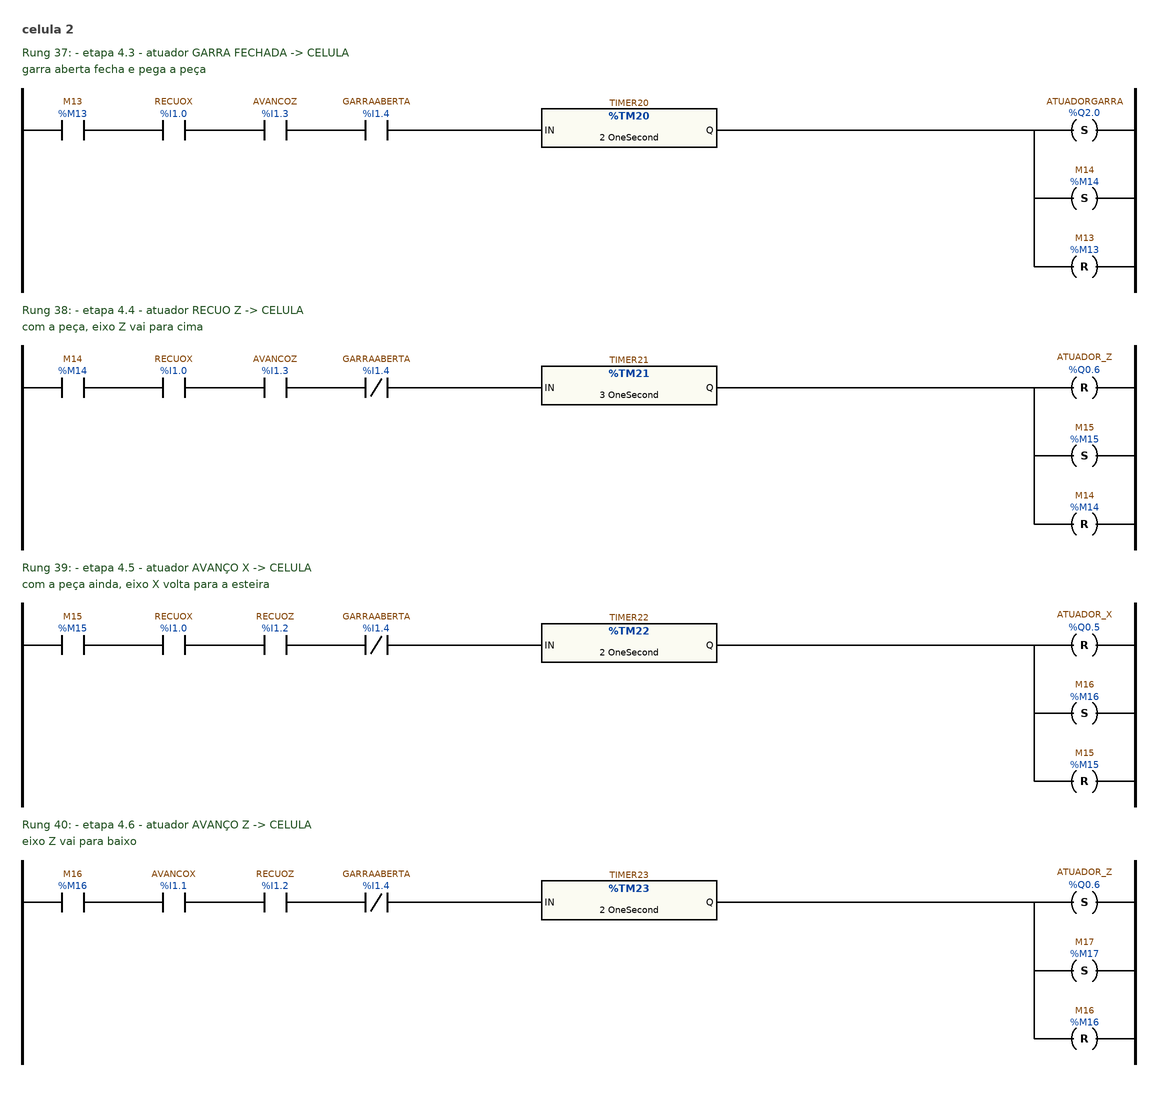

// Rung 37: - etapa 4.3 - atuador GARRA FECHADA -> CELULA
// garra aberta fecha e pega a peça
  BLK %TM20               (* TIMER20 *)
  LD %M13                 (* M13 *)
  AND %I1.0               (* RECUOX *)
  AND %I1.3               (* AVANCOZ *)
  AND %I1.4               (* GARRAABERTA *)
  IN
  OUT_BLK
  LD Q
  S %Q2.0                 (* ATUADORGARRA *)
  S %M14                  (* M14 *)
  R %M13                  (* M13 *)
  END_BLK
  // as ST:
  //   TIMER20(IN := M13 AND RECUOX AND AVANCOZ AND GARRAABERTA);
  //   IF TIMER20.Q THEN ATUADORGARRA := TRUE; END_IF;
  //   IF TIMER20.Q THEN M14 := TRUE; END_IF;
  //   IF TIMER20.Q THEN M13 := FALSE; END_IF;

// Rung 38: - etapa 4.4 - atuador RECUO Z -> CELULA
// com a peça, eixo Z vai para cima
  BLK %TM21               (* TIMER21 *)
  LD %M14                 (* M14 *)
  AND %I1.0               (* RECUOX *)
  AND %I1.3               (* AVANCOZ *)
  ANDN %I1.4              (* GARRAABERTA *)
  IN
  OUT_BLK
  LD Q
  R %Q0.6                 (* ATUADOR_Z *)
  S %M15                  (* M15 *)
  R %M14                  (* M14 *)
  END_BLK
  // as ST:
  //   TIMER21(IN := M14 AND RECUOX AND AVANCOZ AND NOT GARRAABERTA);
  //   IF TIMER21.Q THEN ATUADOR_Z := FALSE; END_IF;
  //   IF TIMER21.Q THEN M15 := TRUE; END_IF;
  //   IF TIMER21.Q THEN M14 := FALSE; END_IF;

// Rung 39: - etapa 4.5 - atuador AVANÇO X -> CELULA
// com a peça ainda, eixo X volta para a esteira
  BLK %TM22               (* TIMER22 *)
  LD %M15                 (* M15 *)
  AND %I1.0               (* RECUOX *)
  AND %I1.2               (* RECUOZ *)
  ANDN %I1.4              (* GARRAABERTA *)
  IN
  OUT_BLK
  LD Q
  R %Q0.5                 (* ATUADOR_X *)
  S %M16                  (* M16 *)
  R %M15                  (* M15 *)
  END_BLK
  // as ST:
  //   TIMER22(IN := M15 AND RECUOX AND RECUOZ AND NOT GARRAABERTA);
  //   IF TIMER22.Q THEN ATUADOR_X := FALSE; END_IF;
  //   IF TIMER22.Q THEN M16 := TRUE; END_IF;
  //   IF TIMER22.Q THEN M15 := FALSE; END_IF;

// Rung 40: - etapa 4.6 - atuador AVANÇO Z -> CELULA
// eixo Z vai para baixo
  BLK %TM23               (* TIMER23 *)
  LD %M16                 (* M16 *)
  AND %I1.1               (* AVANCOX *)
  AND %I1.2               (* RECUOZ *)
  ANDN %I1.4              (* GARRAABERTA *)
  IN
  OUT_BLK
  LD Q
  S %Q0.6                 (* ATUADOR_Z *)
  S %M17                  (* M17 *)
  R %M16                  (* M16 *)
  END_BLK
  // as ST:
  //   TIMER23(IN := M16 AND AVANCOX AND RECUOZ AND NOT GARRAABERTA);
  //   IF TIMER23.Q THEN ATUADOR_Z := TRUE; END_IF;
  //   IF TIMER23.Q THEN M17 := TRUE; END_IF;
  //   IF TIMER23.Q THEN M16 := FALSE; END_IF;

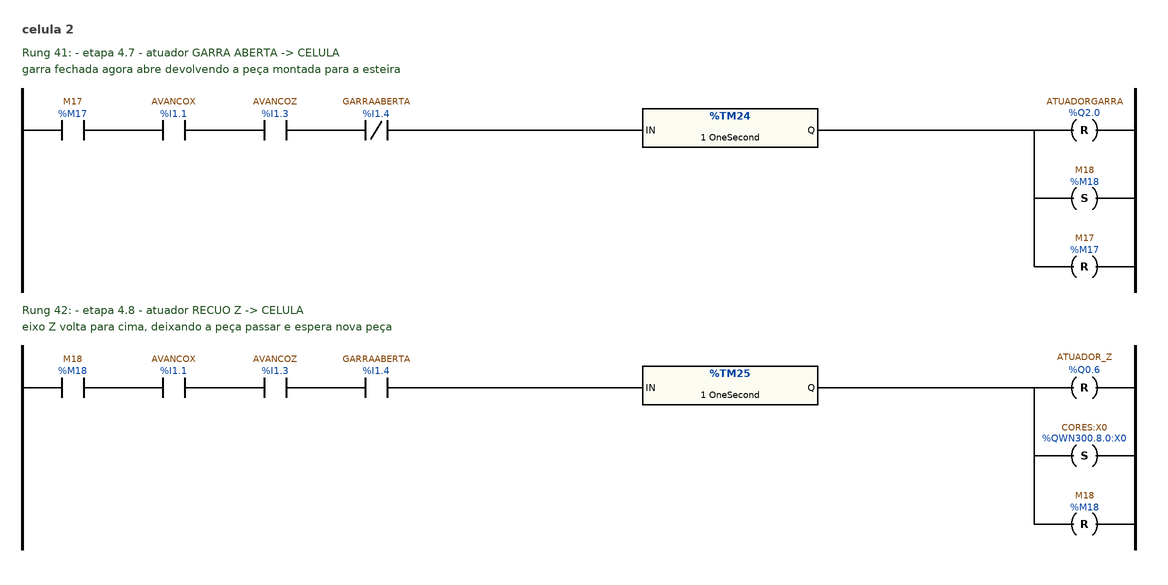

// Rung 41: - etapa 4.7 - atuador GARRA ABERTA -> CELULA
// garra fechada agora abre devolvendo a peça montada para a esteira
  BLK %TM24
  LD %M17                 (* M17 *)
  AND %I1.1               (* AVANCOX *)
  AND %I1.3               (* AVANCOZ *)
  ANDN %I1.4              (* GARRAABERTA *)
  IN
  OUT_BLK
  LD Q
  R %Q2.0                 (* ATUADORGARRA *)
  S %M18                  (* M18 *)
  R %M17                  (* M17 *)
  END_BLK
  // as ST:
  //   %TM24(IN := M17 AND AVANCOX AND AVANCOZ AND NOT GARRAABERTA);
  //   IF %TM24.Q THEN ATUADORGARRA := FALSE; END_IF;
  //   IF %TM24.Q THEN M18 := TRUE; END_IF;
  //   IF %TM24.Q THEN M17 := FALSE; END_IF;

// Rung 42: - etapa 4.8 - atuador RECUO Z -> CELULA
// eixo Z volta para cima, deixando a peça passar e espera nova peça
  BLK %TM25
  LD %M18                 (* M18 *)
  AND %I1.1               (* AVANCOX *)
  AND %I1.3               (* AVANCOZ *)
  AND %I1.4               (* GARRAABERTA *)
  IN
  OUT_BLK
  LD Q
  R %Q0.6                 (* ATUADOR_Z *)
  S %QWN300.8.0:X0        (* CORES *)
  R %M18                  (* M18 *)
  END_BLK
  // as ST:
  //   %TM25(IN := M18 AND AVANCOX AND AVANCOZ AND GARRAABERTA);
  //   IF %TM25.Q THEN ATUADOR_Z := FALSE; END_IF;
  //   IF %TM25.Q THEN CORES:X0 := TRUE; END_IF;
  //   IF %TM25.Q THEN M18 := FALSE; END_IF;

Subroutine robo - clp
  (* SectionNumber=3, Number=1, IsFastTask=true *)

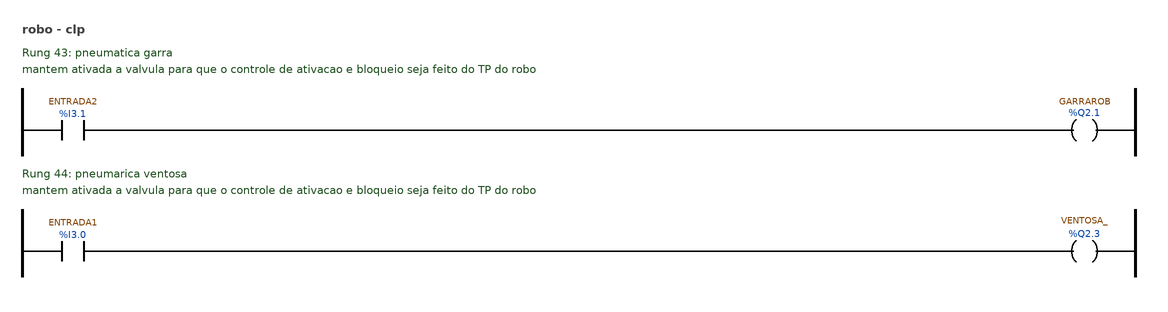

// Rung 43: pneumatica garra
// mantem ativada a valvula para que o controle de ativacao e bloqueio seja feito do TP do robo
  LD %I3.1                (* ENTRADA2 *)
  ST %Q2.1                (* GARRAROB *)
  // as ST:
  //   GARRAROB := ENTRADA2;

// Rung 44: pneumarica ventosa
// mantem ativada a valvula para que o controle de ativacao e bloqueio seja feito do TP do robo
  LD %I3.0                (* ENTRADA1 *)
  ST %Q2.3                (* VENTOSA_ *)
  // as ST:
  //   VENTOSA_ := ENTRADA1;
